KUKA KRL program: ps_ltc_geo_c1.src, ps_ltc_geo_c1.dat

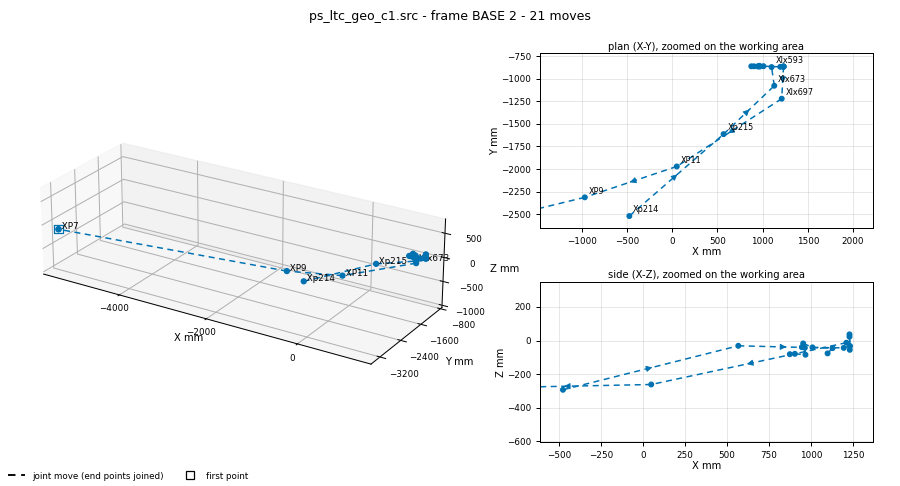
[picture p0: tool path of ps_ltc_geo_c1.src in frame BASE 2, 21 of 24 moves have a stored position in this frame; points joined in program order, loops and branches not executed]
--- ps_ltc_geo_c1.src ---
&ACCESS RVO2
&REL 5
&COMMENT GUN C1 geom Accelo
&PARAM DISKPATH = KRC:\R1\Program
DEF ps_ltc_geo_c1( )
;FOLD INI
;FOLD SPOTTECH INI
USERSPOT(#INIT)
;ENDFOLD (SPOTTECH INI)
;FOLD GRIPPERTECH INI
USER_GRP(0,DUMMY,DUMMY,GDEFAULT)
;ENDFOLD (GRIPPERTECH INI)
  ;FOLD USER INI
    ;Make your modifications here

  ;ENDFOLD (USER INI)
;ENDFOLD (INI)  ;FOLD PTP HOME  Vel= 100 % DEFAULT;%{PE}%V2.2.2,%MKUKATPBASIS,%CMOVE,%VPTP,%P 1:PTP, 2:HOME, 3:, 5:100, 7:DEFAULT

; Caracterização dos meios de produção:
; Versão Atual:
; 12/07/2013 12:00 Name: P13.050-R3 CHANGES: Solda Geometria Accelo
; Pinça C1

chk_w1_wechs_ok ( )         ; CHECK C1

;FOLD PTP P7 CONT Vel=100 % PDAT39 Tool[1]:Gun C1 Base[2]:Accelo;%{PE}%R 8.2.20,%MKUKATPBASIS,%CMOVE,%VPTP,%P 1:PTP, 2:P7, 3:C_DIS, 5:100, 7:PDAT39
$BWDSTART=FALSE
PDAT_ACT=PPDAT39
FDAT_ACT=FP7
BAS(#PTP_PARAMS,100)
PTP XP7 C_DIS
;ENDFOLD

if MaxStandMenge(1) then
  MaxStandmengeErreicht(1)
endif

IF (NOT(GHOST())) THEN
if Elektrodenwechsel(1) then
  e_Fraes1()
endif
ENDIF

;FOLD PTP Pmov_C1_80 CONT Vel=100 % PDAT29 Tool[1]:Gun C1 Base[2]:Accelo;%{PE}%R 8.2.20,%MKUKATPBASIS,%CMOVE,%VPTP,%P 1:PTP, 2:Pmov_C1_80, 3:C_DIS, 5:100, 7:PDAT29
$BWDSTART=FALSE
PDAT_ACT=PPDAT29
FDAT_ACT=FPmov_C1_80
BAS(#PTP_PARAMS,100)
PTP XPmov_C1_80 C_DIS
;ENDFOLD
;FOLD PTP p214 CONT Vel=100 % PDAT21 Tool[1]:Gun C1 Base[2]:Accelo;%{PE}%R 8.2.20,%MKUKATPBASIS,%CMOVE,%VPTP,%P 1:PTP, 2:p214, 3:C_DIS, 5:100, 7:PDAT21
$BWDSTART=FALSE
PDAT_ACT=PPDAT21
FDAT_ACT=Fp214
BAS(#PTP_PARAMS,100)
PTP Xp214 C_DIS
;ENDFOLD

;FOLD OUT 3339 'R3 Soldando' State=TRUE ;%{PE}%R 8.2.20,%MKUKATPBASIS,%COUT,%VOUTX,%P 2:3339, 3:R3 Soldando, 5:TRUE, 6:
$OUT[3339]=TRUE
;ENDFOLD
;FOLD WAIT FOR ( IN 3339 'Aguarda Lib. Soldar Geometria' );%{PE}%R 8.2.20,%MKUKATPBASIS,%CEXT_WAIT_FOR,%VEXT_WAIT_FOR,%P 2:, 4:, 5:$IN, 6:3339, 7:Aguarda Lib. Soldar Geometria, 9:
WAIT FOR  ( $IN[3339] )
;ENDFOLD
;FOLD OUT 3339 'R3 Soldando' State=FALSE ;%{PE}%R 8.2.20,%MKUKATPBASIS,%COUT,%VOUTX,%P 2:3339, 3:R3 Soldando, 5:FALSE, 6:
$OUT[3339]=FALSE
;ENDFOLD
;FOLD OUT 3343 'R3 entregou peça Geo' State=FALSE ;%{PE}%R 8.2.20,%MKUKATPBASIS,%COUT,%VOUTX,%P 2:3343, 3:R3 entregou peça Geo, 5:FALSE, 6:
$OUT[3343]=FALSE
;ENDFOLD
;FOLD OUT 3348 'Fora area GEOBOX' State=FALSE ;%{PE}%R 8.2.20,%MKUKATPBASIS,%COUT,%VOUTX,%P 2:3348, 3:Fora area GEOBOX, 5:FALSE, 6:
$OUT[3348]=FALSE
;ENDFOLD

;FOLD Collision.Monitoring_AREA_1_On ;%{PE}%MKUKATPUSER
COLLSTOP( 7, 1 ) ;not Interrupt-Controlled
;ENDFOLD
;FOLD Collision.Monitoring_AREA_4_On ;%{PE}%MKUKATPUSER
COLLSTOP( 10, 1 ) ;not Interrupt-Controlled
;ENDFOLD

;FOLD PTP p215 CONT Vel=100 % PDAT22 Tool[1]:Gun C1 Base[2]:Accelo;%{PE}%R 8.2.20,%MKUKATPBASIS,%CMOVE,%VPTP,%P 1:PTP, 2:p215, 3:C_DIS, 5:100, 7:PDAT22
$BWDSTART=FALSE
PDAT_ACT=PPDAT22
FDAT_ACT=Fp215
BAS(#PTP_PARAMS,100)
PTP Xp215 C_DIS
;ENDFOLD
;FOLD PTP lx673 CONT Vel=100 % P_OLP5 Tool[1]:Gun C1 Base[2]:Accelo;%{PE}%R 8.2.20,%MKUKATPBASIS,%CMOVE,%VPTP,%P 1:PTP, 2:lx673, 3:C_DIS, 5:100, 7:P_OLP5
$BWDSTART=FALSE
PDAT_ACT=PP_OLP5
FDAT_ACT=Flx673
BAS(#PTP_PARAMS,100)
PTP Xlx673 C_DIS
;ENDFOLD
;FOLD PTP lx593 CONT Vel=100 % P_OLP6 Tool[1]:Gun C1 Base[2]:Accelo;%{PE}%R 8.2.20,%MKUKATPBASIS,%CMOVE,%VPTP,%P 1:PTP, 2:lx593, 3:C_DIS, 5:100, 7:P_OLP6
$BWDSTART=FALSE
PDAT_ACT=PP_OLP6
FDAT_ACT=Flx593
BAS(#PTP_PARAMS,100)
PTP Xlx593 C_DIS
;ENDFOLD
;FOLD PTP P1 CONT Vel=100 % PDAT2 Tool[1]:Gun C1 Base[2]:Accelo;%{PE}%R 8.2.20,%MKUKATPBASIS,%CMOVE,%VPTP,%P 1:PTP, 2:P1, 3:C_DIS, 5:100, 7:PDAT2
$BWDSTART=FALSE
PDAT_ACT=PPDAT2
FDAT_ACT=FP1
BAS(#PTP_PARAMS,100)
PTP XP1 C_DIS
;ENDFOLD

;FOLD ; swp_60_0299;%{PE}%R 5.4.33,%MKUKATPBASIS,%CCOMMENT,%VNORMAL,%P 2:swp_60_0299
;ENDFOLD
;FOLD PTP swp_60_0299 P_OLP7 SPOT Gun=1 RETR CLS PgNo1=1 ACTIVE=1 Tool[1]:Gun C1 Base[2]:Accelo;%{PE}%R 8.2.2,%MKUKATPSPOT,%CSPOT,%VPTP,%P 1:PTP, 2:swp_60_0299, 3:, 5:100, 7:P_OLP7, 10:1, 12:#FIRST, 14:#CLO, 16:1, 18:1, 20:1, 22:0, 24:1, 25:S_OLP1
$BWDSTART=FALSE
PDAT_ACT=PP_OLP7
FDAT_ACT=Fswp_60_0299
BAS(#PTP_PARAMS,PP_OLP7.VEL)
S_ACT.GUN=1
S_ACT.PAIR=SDEFAULT.PAIR
S_ACT.RETR=#CLO
S_ACT.CLO_TM=1
S_ACT.PGNO1=1
S_ACT.PGNO2=SDEFAULT.PGNO2
S_ACT.PRESS1=SDEFAULT.PRESS1
S_ACT.PRESS2=SDEFAULT.PRESS2
S_READY=FALSE
PTP Xswp_60_0299
USERSPOT(#SPOT, S_ACT)
WAIT FOR S_READY
;ENDFOLD

;FOLD ; swp_60_0301;%{PE}%R 8.2.20,%MKUKATPBASIS,%CCOMMENT,%VNORMAL,%P 2:swp_60_0301
;ENDFOLD
;FOLD PTP swp_60_0301 PDAT33 SPOT Gun=1 RETR OPN PgNo1=4 ACTIVE=1 Tool[1]:Gun C1 Base[2]:Accelo;%{PE}%R 8.2.2,%MKUKATPSPOT,%CSPOT,%VPTP,%P 1:PTP, 2:swp_60_0301, 3:, 5:100, 7:PDAT33, 10:1, 12:#FIRST, 14:#OPN, 16:4, 18:1, 20:0, 22:0, 24:1, 25:NORMAL
$BWDSTART=FALSE
PDAT_ACT=PPDAT33
FDAT_ACT=Fswp_60_0301
BAS(#PTP_PARAMS,PPDAT33.VEL)
S_ACT.GUN=1
S_ACT.PAIR=SDEFAULT.PAIR
S_ACT.RETR=#OPN
S_ACT.CLO_TM=1
S_ACT.PGNO1=4
S_ACT.PGNO2=SDEFAULT.PGNO2
S_ACT.PRESS1=SDEFAULT.PRESS1
S_ACT.PRESS2=SDEFAULT.PRESS2
S_READY=FALSE
PTP Xswp_60_0301
USERSPOT(#SPOT, S_ACT)
WAIT FOR S_READY
;ENDFOLD

;FOLD PTP lx692 CONT Vel=100 % P_OLP8 Tool[1]:Gun C1 Base[2]:Accelo;%{PE}%R 8.2.20,%MKUKATPBASIS,%CMOVE,%VPTP,%P 1:PTP, 2:lx692, 3:C_DIS, 5:100, 7:P_OLP8
$BWDSTART=FALSE
PDAT_ACT=PP_OLP8
FDAT_ACT=Flx692
BAS(#PTP_PARAMS,100)
PTP Xlx692 C_DIS
;ENDFOLD
;FOLD PTP P2 CONT Vel=100 % PDAT3 Tool[1]:Gun C1 Base[2]:Accelo;%{PE}%R 8.2.20,%MKUKATPBASIS,%CMOVE,%VPTP,%P 1:PTP, 2:P2, 3:C_DIS, 5:100, 7:PDAT3
$BWDSTART=FALSE
PDAT_ACT=PPDAT3
FDAT_ACT=FP2
BAS(#PTP_PARAMS,100)
PTP XP2 C_DIS
;ENDFOLD

;FOLD ; swp_60_0303;%{PE}%R 8.2.20,%MKUKATPBASIS,%CCOMMENT,%VNORMAL,%P 2:swp_60_0303
;ENDFOLD
;FOLD PTP swp_60_0303 P_OLP29 SPOT Gun=1 RETR CLS PgNo1=2 ACTIVE=1 Tool[1]:Gun C1 Base[2]:Accelo;%{PE}%R 8.2.2,%MKUKATPSPOT,%CSPOT,%VPTP,%P 1:PTP, 2:swp_60_0303, 3:, 5:100, 7:P_OLP29, 10:1, 12:#FIRST, 14:#CLO, 16:2, 18:1, 20:1, 22:0, 24:1, 25:S_OLP2
$BWDSTART=FALSE
PDAT_ACT=PP_OLP29
FDAT_ACT=Fswp_60_0303
BAS(#PTP_PARAMS,PP_OLP29.VEL)
S_ACT.GUN=1
S_ACT.PAIR=SDEFAULT.PAIR
S_ACT.RETR=#CLO
S_ACT.CLO_TM=1
S_ACT.PGNO1=2
S_ACT.PGNO2=SDEFAULT.PGNO2
S_ACT.PRESS1=SDEFAULT.PRESS1
S_ACT.PRESS2=SDEFAULT.PRESS2
S_READY=FALSE
PTP Xswp_60_0303
USERSPOT(#SPOT, S_ACT)
WAIT FOR S_READY
;ENDFOLD

;FOLD ; swp_0305;%{PE}%R 8.2.20,%MKUKATPBASIS,%CCOMMENT,%VNORMAL,%P 2:swp_0305
;ENDFOLD
;FOLD PTP swp_60_0305 PDAT34 SPOT Gun=1 RETR OPN PgNo1=5 ACTIVE=1 Tool[1]:Gun C1 Base[2]:Accelo;%{PE}%R 8.2.2,%MKUKATPSPOT,%CSPOT,%VPTP,%P 1:PTP, 2:swp_60_0305, 3:, 5:100, 7:PDAT34, 10:1, 12:#FIRST, 14:#OPN, 16:5, 18:1, 20:0, 22:0, 24:1, 25:NORMAL
$BWDSTART=FALSE
PDAT_ACT=PPDAT34
FDAT_ACT=Fswp_60_0305
BAS(#PTP_PARAMS,PPDAT34.VEL)
S_ACT.GUN=1
S_ACT.PAIR=SDEFAULT.PAIR
S_ACT.RETR=#OPN
S_ACT.CLO_TM=1
S_ACT.PGNO1=5
S_ACT.PGNO2=SDEFAULT.PGNO2
S_ACT.PRESS1=SDEFAULT.PRESS1
S_ACT.PRESS2=SDEFAULT.PRESS2
S_READY=FALSE
PTP Xswp_60_0305
USERSPOT(#SPOT, S_ACT)
WAIT FOR S_READY
;ENDFOLD

;FOLD PTP lx693 CONT Vel=100 % P_OLP10 Tool[1]:Gun C1 Base[2]:Accelo;%{PE}%R 8.2.20,%MKUKATPBASIS,%CMOVE,%VPTP,%P 1:PTP, 2:lx693, 3:C_DIS, 5:100, 7:P_OLP10
$BWDSTART=FALSE
PDAT_ACT=PP_OLP10
FDAT_ACT=Flx693
BAS(#PTP_PARAMS,100)
PTP Xlx693 C_DIS
;ENDFOLD
;FOLD PTP lx694 CONT Vel=100 % P_OLP11 Tool[1]:Gun C1 Base[2]:Accelo;%{PE}%R 8.2.20,%MKUKATPBASIS,%CMOVE,%VPTP,%P 1:PTP, 2:lx694, 3:C_DIS, 5:100, 7:P_OLP11
$BWDSTART=FALSE
PDAT_ACT=PP_OLP11
FDAT_ACT=Flx694
BAS(#PTP_PARAMS,100)
PTP Xlx694 C_DIS
;ENDFOLD
;FOLD PTP lx695 CONT Vel=100 % P_OLP12 Tool[1]:Gun C1 Base[2]:Accelo;%{PE}%R 8.2.20,%MKUKATPBASIS,%CMOVE,%VPTP,%P 1:PTP, 2:lx695, 3:C_DIS, 5:100, 7:P_OLP12
$BWDSTART=FALSE
PDAT_ACT=PP_OLP12
FDAT_ACT=Flx695
BAS(#PTP_PARAMS,100)
PTP Xlx695 C_DIS
;ENDFOLD

;FOLD ; swp_60_0311;%{PE}%R 5.4.33,%MKUKATPBASIS,%CCOMMENT,%VNORMAL,%P 2:swp_60_0311
;ENDFOLD
;FOLD PTP swp_60_0311 P_OLP13 SPOT Gun=1 RETR CLS PgNo1=3 ACTIVE=1 Tool[1]:Gun C1 Base[2]:Accelo;%{PE}%R 8.2.2,%MKUKATPSPOT,%CSPOT,%VPTP,%P 1:PTP, 2:swp_60_0311, 3:, 5:100, 7:P_OLP13, 10:1, 12:#FIRST, 14:#CLO, 16:3, 18:1, 20:1, 22:0, 24:1, 25:S_OLP3
$BWDSTART=FALSE
PDAT_ACT=PP_OLP13
FDAT_ACT=Fswp_60_0311
BAS(#PTP_PARAMS,PP_OLP13.VEL)
S_ACT.GUN=1
S_ACT.PAIR=SDEFAULT.PAIR
S_ACT.RETR=#CLO
S_ACT.CLO_TM=1
S_ACT.PGNO1=3
S_ACT.PGNO2=SDEFAULT.PGNO2
S_ACT.PRESS1=SDEFAULT.PRESS1
S_ACT.PRESS2=SDEFAULT.PRESS2
S_READY=FALSE
PTP Xswp_60_0311
USERSPOT(#SPOT, S_ACT)
WAIT FOR S_READY
;ENDFOLD

;FOLD ; swp_60_0313;%{PE}%R 8.2.20,%MKUKATPBASIS,%CCOMMENT,%VNORMAL,%P 2:swp_60_0313
;ENDFOLD
;FOLD PTP swp_60_0313 PDAT35 SPOT Gun=1 RETR OPN PgNo1=6 ACTIVE=1 Tool[1]:Gun C1 Base[2]:Accelo;%{PE}%R 8.2.2,%MKUKATPSPOT,%CSPOT,%VPTP,%P 1:PTP, 2:swp_60_0313, 3:, 5:100, 7:PDAT35, 10:1, 12:#FIRST, 14:#OPN, 16:6, 18:1, 20:0, 22:0, 24:1, 25:NORMAL
$BWDSTART=FALSE
PDAT_ACT=PPDAT35
FDAT_ACT=Fswp_60_0313
BAS(#PTP_PARAMS,PPDAT35.VEL)
S_ACT.GUN=1
S_ACT.PAIR=SDEFAULT.PAIR
S_ACT.RETR=#OPN
S_ACT.CLO_TM=1
S_ACT.PGNO1=6
S_ACT.PGNO2=SDEFAULT.PGNO2
S_ACT.PRESS1=SDEFAULT.PRESS1
S_ACT.PRESS2=SDEFAULT.PRESS2
S_READY=FALSE
PTP Xswp_60_0313
USERSPOT(#SPOT, S_ACT)
WAIT FOR S_READY
;ENDFOLD

;FOLD PTP lx696 CONT Vel=100 % P_OLP14 Tool[1]:Gun C1 Base[2]:Accelo;%{PE}%R 8.2.20,%MKUKATPBASIS,%CMOVE,%VPTP,%P 1:PTP, 2:lx696, 3:C_DIS, 5:100, 7:P_OLP14
$BWDSTART=FALSE
PDAT_ACT=PP_OLP14
FDAT_ACT=Flx696
BAS(#PTP_PARAMS,100)
PTP Xlx696 C_DIS
;ENDFOLD
;FOLD PTP lx697 CONT Vel=100 % P_OLP15 Tool[1]:Gun C1 Base[2]:Accelo;%{PE}%R 8.2.20,%MKUKATPBASIS,%CMOVE,%VPTP,%P 1:PTP, 2:lx697, 3:C_DIS, 5:100, 7:P_OLP15
$BWDSTART=FALSE
PDAT_ACT=PP_OLP15
FDAT_ACT=Flx697
BAS(#PTP_PARAMS,100)
PTP Xlx697 C_DIS
;ENDFOLD
;FOLD PTP P11 Vel=100 % PDAT43 Tool[1]:Gun C1 Base[2]:Accelo;%{PE}%R 8.2.20,%MKUKATPBASIS,%CMOVE,%VPTP,%P 1:PTP, 2:P11, 3:, 5:100, 7:PDAT43
$BWDSTART=FALSE
PDAT_ACT=PPDAT43
FDAT_ACT=FP11
BAS(#PTP_PARAMS,100)
PTP XP11
;ENDFOLD

;FOLD Collision.Monitoring_AREA_4_Off . ;%{PE}%MKUKATPUSER
COLLSTOP( 10, 2+0 )
;ENDFOLD

;FOLD PTP P9 Vel=100 % PDAT41 Tool[1]:Gun C1 Base[2]:Accelo;%{PE}%R 8.2.20,%MKUKATPBASIS,%CMOVE,%VPTP,%P 1:PTP, 2:P9, 3:, 5:100, 7:PDAT41
$BWDSTART=FALSE
PDAT_ACT=PPDAT41
FDAT_ACT=FP9
BAS(#PTP_PARAMS,100)
PTP XP9
;ENDFOLD

;FOLD Collision.Monitoring_AREA_1_Off . ;%{PE}%MKUKATPUSER
COLLSTOP( 7, 2+0 )
;ENDFOLD
;FOLD OUT 3348 'Fora area GEOBOX' State=TRUE ;%{PE}%R 8.2.20,%MKUKATPBASIS,%COUT,%VOUTX,%P 2:3348, 3:Fora area GEOBOX, 5:TRUE, 6:
$OUT[3348]=TRUE
;ENDFOLD

;FOLD PTP lx33 CONT Vel=100 % P_OLP22 Tool[1]:Gun C1 Base[2]:Accelo;%{PE}%R 8.2.20,%MKUKATPBASIS,%CMOVE,%VPTP,%P 1:PTP, 2:lx33, 3:C_DIS, 5:100, 7:P_OLP22
$BWDSTART=FALSE
PDAT_ACT=PP_OLP22
FDAT_ACT=Flx33
BAS(#PTP_PARAMS,100)
PTP Xlx33 C_DIS
;ENDFOLD

IF (NOT(GHOST())) THEN
if FraesAnf(1) then
  f_fraes1()
endif
ENDIF

;FOLD PTP P8 CONT Vel=100 % PDAT40 Tool[1]:Gun C1 Base[2]:Accelo;%{PE}%R 8.2.20,%MKUKATPBASIS,%CMOVE,%VPTP,%P 1:PTP, 2:P8, 3:C_DIS, 5:100, 7:PDAT40
$BWDSTART=FALSE
PDAT_ACT=PPDAT40
FDAT_ACT=FP8
BAS(#PTP_PARAMS,100)
PTP XP8 C_DIS
;ENDFOLD

END

--- ps_ltc_geo_c1.dat ---
&ACCESS RVO2
&REL 5
&COMMENT GUN C1 geom Accelo
&PARAM DISKPATH = KRC:\R1\Program
DEFDAT  ps_ltc_geo_c1
;FOLD EXTERNAL DECLARATIONS;%{PE}%MKUKATPBASIS,%CEXT,%VCOMMON,%P
;FOLD GRIPPERTECH EXT
EXT  H50 (INT  :IN,INT  :IN,INT  :IN,GRP_TYP  :IN )
;ENDFOLD (GRIPPERTECH EXT)
;FOLD SPOTTECH EXT
EXT  USERSPOT (S_COMMAND  :IN,SPOT_TYPE  :IN )
;ENDFOLD (SPOTTECH EXT)
;FOLD BASISTECH EXT;%{PE}%MKUKATPBASIS,%CEXT,%VEXT,%P
EXT  BAS (BAS_COMMAND  :IN,REAL  :IN )
DECL INT SUCCESS
;ENDFOLD (BASISTECH EXT)
;FOLD USER EXT;%{E}%MKUKATPUSER,%CEXT,%VEXT,%P
;Make your modifications here

;ENDFOLD (USER EXT)
;ENDFOLD (EXTERNAL DECLARATIONS)
;# ============ START PATH : swp_p13050r3_ltc_geo_c1 =============
DECL FDAT Flx673={TOOL_NO 1,BASE_NO 2,IPO_FRAME #BASE,POINT2[] " "}
DECL PDAT PP_OLP5={VEL 100.0,ACC 100.0,APO_DIST 100.0,APO_MODE #CDIS}
DECL E6POS Xlx673={X 1127.99402,Y -1078.20105,Z -45.247509,A 177.553497,B -1.23780203,C -81.5183105,S 2,T 11,E1 5590.04492,E2 0.0,E3 0.0,E4 0.0,E5 0.0,E6 0.0}
DECL FDAT Flx593={TOOL_NO 1,BASE_NO 2,IPO_FRAME #BASE,POINT2[] " "}
DECL PDAT PP_OLP6={VEL 100.0,ACC 100.0,APO_DIST 100.0,APO_MODE #CDIS}
DECL E6POS Xlx593={X 1098.53894,Y -871.950317,Z -76.444603,A 177.514999,B -1.16095197,C -79.743309,S 2,T 11,E1 5590.04492,E2 0.0,E3 0.0,E4 0.0,E5 0.0,E6 0.0}
DECL FDAT Fswp_60_0299={TOOL_NO 1,BASE_NO 2,IPO_FRAME #BASE,POINT2[] " "}
DECL PDAT PP_OLP7={VEL 100.0,ACC 100.0,APO_DIST 0.0}
DECL SPOT_TYPE SS_OLP1={GUN 1,PAIR #FIRST,RETR #OPN,CLO_TM 0,PGNO1 1,PRESS1 1.0,PGNO2 0,PRESS2 0.0}
DECL E6POS Xswp_60_0299={X 874.041077,Y -863.023682,Z -81.2979202,A 177.433105,B -0.103535101,C -83.8159027,S 2,T 11,E1 5590.04297,E2 0.0,E3 0.0,E4 0.0,E5 0.0,E6 0.0}
DECL FDAT Flx692={TOOL_NO 1,BASE_NO 2,IPO_FRAME #BASE,POINT2[] " "}
DECL PDAT PP_OLP8={VEL 100.0,ACC 100.0,APO_DIST 100.0,APO_MODE #CDIS}
DECL E6POS Xlx692={X 967.02063,Y -865.732727,Z -84.5335007,A 177.432999,B 3.48430109,C -79.9825211,S 2,T 11,E1 5590.04199,E2 0.0,E3 0.0,E4 0.0,E5 0.0,E6 0.0}
DECL FDAT Fswp_60_0303={TOOL_NO 1,BASE_NO 2,IPO_FRAME #BASE,POINT2[] " "}
DECL SPOT_TYPE SS_OLP2={GUN 1,PAIR #FIRST,RETR #OPN,CLO_TM 0,PGNO1 1,PRESS1 1.0,PGNO2 0,PRESS2 0.0}
DECL E6POS Xswp_60_0303={X 945.597107,Y -864.208923,Z -39.588501,A 177.035004,B -10.4853096,C -81.7657623,S 2,T 11,E1 5590.04199,E2 0.0,E3 0.0,E4 0.0,E5 0.0,E6 0.0}
DECL FDAT Flx693={TOOL_NO 1,BASE_NO 2,IPO_FRAME #BASE,POINT2[] " "}
DECL PDAT PP_OLP10={VEL 100.0,ACC 100.0,APO_DIST 100.0,APO_MODE #CDIS}
DECL E6POS Xlx693={X 1008.59399,Y -862.025574,Z -40.7261887,A 177.0354,B -10.4855804,C -81.7657623,S 2,T 11,E1 5590.04199,E2 0.0,E3 0.0,E4 0.0,E5 0.0,E6 0.0}
DECL FDAT Flx694={TOOL_NO 1,BASE_NO 2,IPO_FRAME #BASE,POINT2[] " "}
DECL PDAT PP_OLP11={VEL 100.0,ACC 100.0,APO_DIST 100.0,APO_MODE #CDIS}
DECL E6POS Xlx694={X 1194.74805,Y -868.942688,Z -43.8955116,A 177.039093,B -10.4863796,C -81.7690735,S 2,T 11,E1 5590.04199,E2 0.0,E3 0.0,E4 0.0,E5 0.0,E6 0.0}
DECL FDAT Flx695={TOOL_NO 1,BASE_NO 2,IPO_FRAME #BASE,POINT2[] " "}
DECL PDAT PP_OLP12={VEL 100.0,ACC 100.0,APO_DIST 100.0,APO_MODE #CDIS}
DECL E6POS Xlx695={X 1232.04395,Y -868.190613,Z -32.9681587,A 176.107803,B -16.6657391,C -81.5498734,S 2,T 11,E1 5590.04199,E2 0.0,E3 0.0,E4 0.0,E5 0.0,E6 0.0}
DECL FDAT Fswp_60_0311={TOOL_NO 1,BASE_NO 2,IPO_FRAME #BASE,POINT2[] " "}
DECL PDAT PP_OLP13={VEL 100.0,ACC 100.0,APO_DIST 0.0}
DECL SPOT_TYPE SS_OLP3={GUN 1,PAIR #FIRST,RETR #OPN,CLO_TM 0,PGNO1 1,PRESS1 1.0,PGNO2 0,PRESS2 0.0}
DECL E6POS Xswp_60_0311={X 1228.85303,Y -865.706909,Z 36.6585388,A -179.803894,B -38.7357712,C -88.0000916,S 2,T 11,E1 5590.04102,E2 0.0,E3 0.0,E4 0.0,E5 0.0,E6 0.0}
DECL FDAT Flx696={TOOL_NO 1,BASE_NO 2,IPO_FRAME #BASE,POINT2[] " "}
DECL PDAT PP_OLP14={VEL 100.0,ACC 100.0,APO_DIST 50.0,APO_MODE #CDIS}
DECL E6POS Xlx696={X 1230.51794,Y -864.94281,Z -55.2660408,A 176.131195,B -16.5310497,C -81.61409,S 2,T 11,E1 5590.04199,E2 0.0,E3 0.0,E4 0.0,E5 0.0,E6 0.0}
DECL FDAT Flx697={TOOL_NO 1,BASE_NO 2,IPO_FRAME #BASE,POINT2[] " "}
DECL PDAT PP_OLP15={VEL 100.0,ACC 100.0,APO_DIST 100.0,APO_MODE #CDIS}
DECL E6POS Xlx697={X 1210.396,Y -1221.43799,Z -13.2171497,A 168.579498,B -15.2477703,C -79.5598297,S 2,T 11,E1 5590.04199,E2 0.0,E3 0.0,E4 0.0,E5 0.0,E6 0.0}
DECL BASIS_SUGG_T LAST_BASIS={POINT1[] "P0                      ",POINT2[] "P0                      ",CP_PARAMS[] "CPDAT0                  ",PTP_PARAMS[] "PDAT0                   ",CONT[] "                        ",CP_VEL[] "2.0                     ",PTP_VEL[] " 100                    ",SYNC_PARAMS[] "SYNCDAT                 ",SPL_NAME[] "S0                      "}
DECL SPOT_SUGG_T LAST_SPOT={GUN[] "1                       ",RETR_CMD[] "#OPN                    ",CHOISE[] "#FIRST                  ",CLO_TM[] "1                       ",PGNO1[] "4                       ",PRESS1[] "0                       ",PGNO2[] "1                       ",PRESS2[] "0                       ",SPOT_PARAMS[] "NORMAL                  "}
DECL E6POS XP1={X 1853.93201,Y -7469.54102,Z 1558.43005,A 87.4294891,B 3.4838469,C -79.9745712,S 2,T 11,E1 5590.04199,E2 0.0,E3 0.0,E4 0.0,E5 0.0,E6 0.0}
DECL FDAT FP1={TOOL_NO 1,BASE_NO 0,IPO_FRAME #BASE,POINT2[] " ",TQ_STATE FALSE}
DECL PDAT PPDAT2={VEL 100.0,ACC 100.0,APO_DIST 100.0,APO_MODE #CDIS}
DECL E6POS XP2={X 963.036682,Y -857.634888,Z -43.4037209,A 177.115402,B -6.82887316,C -81.6067505,S 2,T 11,E1 5590.04199,E2 0.0,E3 0.0,E4 0.0,E5 0.0,E6 0.0}
DECL FDAT FP2={TOOL_NO 1,BASE_NO 2,IPO_FRAME #BASE,POINT2[] " ",TQ_STATE FALSE}
DECL PDAT PPDAT3={VEL 100.0,ACC 100.0,APO_DIST 100.0,APO_MODE #CDIS}
DECL E6POS XP214={X -474.976807,Y -2519.66797,Z -292.991394,A 152.031296,B 2.67392898,C -27.66502,S 2,T 11,E1 4006.78809,E2 0.0,E3 0.0,E4 0.0,E5 0.0,E6 0.0}
DECL FDAT Fp214={TOOL_NO 1,BASE_NO 2,IPO_FRAME #BASE,POINT2[] " ",TQ_STATE FALSE}
DECL PDAT PPDAT21={VEL 100.0,ACC 100.0,APO_DIST 100.0,APO_MODE #CDIS}
DECL E6POS XP215={X 567.599121,Y -1613.47205,Z -31.5026302,A -178.177399,B -5.01841116,C -73.1850433,S 2,T 11,E1 5076.10303,E2 0.0,E3 0.0,E4 0.0,E5 0.0,E6 0.0}
DECL FDAT Fp215={TOOL_NO 1,BASE_NO 2,IPO_FRAME #BASE,POINT2[] " ",TQ_STATE FALSE}
DECL PDAT PPDAT22={VEL 100.0,ACC 100.0,APO_DIST 100.0,APO_MODE #CDIS}
DECL PDAT PPDAT29={VEL 100.0,ACC 100.0,APO_DIST 100.0,APO_MODE #CDIS}
DECL E6POS XPmov_C1_80={X -3984.38403,Y -2519.66699,Z -155.263702,A 152.031296,B 2.67380309,C -27.6649609,S 2,T 11,E1 293.084106,E2 0.0,E3 0.0,E4 0.0,E5 0.0,E6 0.0}
DECL FDAT FPmov_C1_80={TOOL_NO 1,BASE_NO 1,IPO_FRAME #BASE,POINT2[] " ",TQ_STATE FALSE}
DECL PDAT PP_OLP22={VEL 100.0,ACC 100.0,APO_DIST 0.0,APO_MODE #CDIS}
DECL E6POS Xlx33={X -5502.85498,Y -3417.39307,Z -55.4117088,A 134.611603,B 6.01144505,C -0.767602026,S 2,T 10,E1 297.920105,E2 0.0,E3 0.0,E4 0.0,E5 0.0,E6 0.0}
DECL FDAT Flx33={TOOL_NO 1,BASE_NO 2,IPO_FRAME #BASE,POINT2[] " ",TQ_STATE FALSE}
DECL E6POS Xswp_60_0305={X 953.553589,Y -863.275513,Z -17.3715096,A 177.2146,B -13.4707003,C -82.5131912,S 2,T 11,E1 5590.04102,E2 0.0,E3 0.0,E4 0.0,E5 0.0,E6 0.0}
DECL FDAT Fswp_60_0305={TOOL_NO 1,BASE_NO 2,IPO_FRAME #BASE,POINT2[] " "}
DECL PDAT PPDAT33={VEL 100.0,ACC 100.0,APO_DIST 100.0}
DECL PDAT PPDAT34={VEL 100.0,ACC 100.0,APO_DIST 100.0}
DECL PDAT PPDAT35={VEL 100.0,ACC 100.0,APO_DIST 100.0}
DECL E6POS XP7={X -5500.30908,Y -3416.72412,Z -55.3835411,A 125.481903,B 5.81504917,C -1.709777,S 2,T 10,E1 299.244598,E2 0.0,E3 0.0,E4 0.0,E5 0.0,E6 0.0}
DECL FDAT FP7={TOOL_NO 1,BASE_NO 2,IPO_FRAME #BASE,POINT2[] " ",TQ_STATE FALSE}
DECL PDAT PPDAT39={VEL 100.0,ACC 100.0,APO_DIST 20.0,APO_MODE #CDIS}
DECL E6POS XP8={X 111.676804,Y 1355.45203,Z 1650.13196,A -97.9474106,B 21.7212791,C -2.70396805,S 2,T 10,E1 296.308685,E2 0.0,E3 0.0,E4 0.0,E5 0.0,E6 0.0}
DECL FDAT FP8={TOOL_NO 1,BASE_NO 0,IPO_FRAME #BASE,POINT2[] " ",TQ_STATE FALSE}
DECL PDAT PPDAT40={VEL 100.0,ACC 100.0,APO_DIST 25.0,APO_MODE #CDIS}
DECL PDAT PP_OLP29={VEL 100.0,ACC 100.0,APO_DIST 0.0}
DECL E6POS XP9={X -967.743286,Y -2312.36694,Z -282.115814,A -168.154007,B -10.7438297,C -39.5715408,S 2,T 11,E1 4107.69092,E2 0.0,E3 0.0,E4 0.0,E5 0.0,E6 0.0}
DECL FDAT FP9={TOOL_NO 1,BASE_NO 2,IPO_FRAME #BASE,POINT2[] " ",TQ_STATE FALSE}
DECL PDAT PPDAT41={VEL 100.0,ACC 100.0,APO_DIST 0.0,APO_MODE #CDIS}
DECL E6POS Xswp_60_0301={X 903.826599,Y -863.021484,Z -79.1251373,A 177.434799,B -0.127913296,C -84.3507767,S 2,T 11,E1 5590.04199,E2 0.0,E3 0.0,E4 0.0,E5 0.0,E6 0.0}
DECL FDAT Fswp_60_0301={TOOL_NO 1,BASE_NO 2,IPO_FRAME #BASE,POINT2[] " ",TQ_STATE FALSE}
DECL E6POS Xswp_60_0313={X 1228.84094,Y -865.707275,Z 22.5872402,A -179.802597,B -38.7351418,C -88.0015869,S 2,T 11,E1 5590.04102,E2 0.0,E3 0.0,E4 0.0,E5 0.0,E6 0.0}
DECL FDAT Fswp_60_0313={TOOL_NO 1,BASE_NO 2,IPO_FRAME #BASE,POINT2[] " ",TQ_STATE FALSE}
DECL E6POS XP11={X 49.6881294,Y -1970.96997,Z -261.569794,A -174.3535,B 4.73328018,C -45.3660011,S 2,T 11,E1 4614.18799,E2 0.0,E3 0.0,E4 0.0,E5 0.0,E6 0.0}
DECL FDAT FP11={TOOL_NO 1,BASE_NO 2,IPO_FRAME #BASE,POINT2[] " ",TQ_STATE FALSE}
DECL PDAT PPDAT43={VEL 100.0,ACC 100.0,APO_DIST 50.0,APO_MODE #CDIS}
ENDDAT
